Fanuc TP program (LS listing): FANUC_JOGJ.ls

/PROG  FANUC_JOGJ
/ATTR
OWNER		= MNEDITOR;
COMMENT		= "Stream joint jog";
PROG_SIZE	= 0;
CREATE		= DATE 26-04-16  TIME 10:00:00;
MODIFIED	= DATE 26-04-16  TIME 10:00:00;
FILE_NAME	= ;
VERSION		= 0;
LINE_COUNT	= 113;
MEMORY_SIZE	= 0;
PROTECT		= READ_WRITE;
TCD:  STACK_SIZE	= 0,
      TASK_PRIORITY	= 50,
      TIME_SLICE	= 0,
      BUSY_LAMP_OFF	= 0,
      ABORT_REQUEST	= 0,
      PAUSE_REQUEST	= 0;
DEFAULT_GROUP	= 1,*,*,*,*;
CONTROL_CODE	= 00000000 00000000;
/MN
   1:  R[85]=0 ;
   2:  UFRAME_NUM=0 ;
   3:  UTOOL_NUM=1 ;
   4:  R[81]=0 ;
   5:  R[82]=0 ;
   6:  R[84]=0 ;
   7:  CALL LOADJOGBUF ;
   8:  IF R[84]<>1,JMP LBL[99] ;
   9:  LBL[1] ;
  10:  IF R[80]=1,JMP LBL[10] ;
  11:  IF R[81]>=R[82],JMP LBL[99] ;
  12:  LBL[10] ;
  13:  J PR[20] R[17]% CNT50 ;
  14:  R[81]=R[81]+1 ;
  15:  IF R[80]=1,JMP LBL[11] ;
  16:  IF R[81]>=R[82],JMP LBL[99] ;
  17:  LBL[11] ;
  18:  J PR[21] R[17]% CNT50 ;
  19:  R[81]=R[81]+1 ;
  20:  IF R[80]=1,JMP LBL[12] ;
  21:  IF R[81]>=R[82],JMP LBL[99] ;
  22:  LBL[12] ;
  23:  J PR[22] R[17]% CNT50 ;
  24:  R[81]=R[81]+1 ;
  25:  IF R[80]=1,JMP LBL[13] ;
  26:  IF R[81]>=R[82],JMP LBL[99] ;
  27:  LBL[13] ;
  28:  J PR[23] R[17]% CNT50 ;
  29:  R[81]=R[81]+1 ;
  30:  IF R[80]=1,JMP LBL[14] ;
  31:  IF R[81]>=R[82],JMP LBL[99] ;
  32:  LBL[14] ;
  33:  J PR[24] R[17]% CNT50 ;
  34:  R[81]=R[81]+1 ;
  35:  IF R[80]=1,JMP LBL[15] ;
  36:  IF R[81]>=R[82],JMP LBL[99] ;
  37:  LBL[15] ;
  38:  J PR[25] R[17]% CNT50 ;
  39:  R[81]=R[81]+1 ;
  40:  IF R[80]=1,JMP LBL[16] ;
  41:  IF R[81]>=R[82],JMP LBL[99] ;
  42:  LBL[16] ;
  43:  J PR[26] R[17]% CNT50 ;
  44:  R[81]=R[81]+1 ;
  45:  IF R[80]=1,JMP LBL[17] ;
  46:  IF R[81]>=R[82],JMP LBL[99] ;
  47:  LBL[17] ;
  48:  J PR[27] R[17]% CNT50 ;
  49:  R[81]=R[81]+1 ;
  50:  IF R[80]=1,JMP LBL[18] ;
  51:  IF R[81]>=R[82],JMP LBL[99] ;
  52:  LBL[18] ;
  53:  J PR[28] R[17]% CNT50 ;
  54:  R[81]=R[81]+1 ;
  55:  IF R[80]=1,JMP LBL[19] ;
  56:  IF R[81]>=R[82],JMP LBL[99] ;
  57:  LBL[19] ;
  58:  J PR[29] R[17]% CNT50 ;
  59:  R[81]=R[81]+1 ;
  60:  IF R[80]=1,JMP LBL[20] ;
  61:  IF R[81]>=R[82],JMP LBL[99] ;
  62:  LBL[20] ;
  63:  J PR[30] R[17]% CNT50 ;
  64:  R[81]=R[81]+1 ;
  65:  IF R[80]=1,JMP LBL[21] ;
  66:  IF R[81]>=R[82],JMP LBL[99] ;
  67:  LBL[21] ;
  68:  J PR[31] R[17]% CNT50 ;
  69:  R[81]=R[81]+1 ;
  70:  IF R[80]=1,JMP LBL[22] ;
  71:  IF R[81]>=R[82],JMP LBL[99] ;
  72:  LBL[22] ;
  73:  J PR[32] R[17]% CNT50 ;
  74:  R[81]=R[81]+1 ;
  75:  IF R[80]=1,JMP LBL[23] ;
  76:  IF R[81]>=R[82],JMP LBL[99] ;
  77:  LBL[23] ;
  78:  J PR[33] R[17]% CNT50 ;
  79:  R[81]=R[81]+1 ;
  80:  IF R[80]=1,JMP LBL[24] ;
  81:  IF R[81]>=R[82],JMP LBL[99] ;
  82:  LBL[24] ;
  83:  J PR[34] R[17]% CNT50 ;
  84:  R[81]=R[81]+1 ;
  85:  IF R[80]=1,JMP LBL[25] ;
  86:  IF R[81]>=R[82],JMP LBL[99] ;
  87:  LBL[25] ;
  88:  J PR[35] R[17]% CNT50 ;
  89:  R[81]=R[81]+1 ;
  90:  IF R[80]=1,JMP LBL[26] ;
  91:  IF R[81]>=R[82],JMP LBL[99] ;
  92:  LBL[26] ;
  93:  J PR[36] R[17]% CNT50 ;
  94:  R[81]=R[81]+1 ;
  95:  IF R[80]=1,JMP LBL[27] ;
  96:  IF R[81]>=R[82],JMP LBL[99] ;
  97:  LBL[27] ;
  98:  J PR[37] R[17]% CNT50 ;
  99:  R[81]=R[81]+1 ;
 100:  IF R[80]=1,JMP LBL[28] ;
 101:  IF R[81]>=R[82],JMP LBL[99] ;
 102:  LBL[28] ;
 103:  J PR[38] R[17]% CNT50 ;
 104:  R[81]=R[81]+1 ;
 105:  IF R[80]=1,JMP LBL[29] ;
 106:  IF R[81]>=R[82],JMP LBL[99] ;
 107:  LBL[29] ;
 108:  J PR[39] R[17]% CNT50 ;
 109:  R[81]=R[81]+1 ;
 110:  JMP LBL[1] ;
 111:  LBL[99] ;
 112:  R[85]=1 ;
 113:  END ;
/POS
/END
